{attribute 'TcGenerated'}
// This function has been automatically generated from the project information.
VAR_GLOBAL CONSTANT
    {attribute 'const_non_replaced'}
    {attribute 'linkalways'}
    stLibVersion_lcls_plc_tmo_vac : ST_LibVersion := (iMajor := 1, iMinor := 1, iBuild := 0, iRevision := 0, sVersion := '1.1.0');
END_VAR

(* stored: Version 1.1.0.1, ProductVersion 3.1.4022.18
   GVL Global_Version: Id d9b1849f-17dc-42be-8bc8-a6a59c08eba9 *)
